FUNCTION_BLOCK FB_EstacionRestaurar_SFC
VAR_INPUT
    // SFC-Flags
    SFCPause: BOOL;
    SFCReset: BOOL;
    
    // Indicadores de sincronizacion
    Benido: BOOL := TRUE;
    Ejecuta: BOOL;
    
    // Entradas
    RechazadorDetras: BOOL; // Sobre el pale
    ManipuladorMedio: BOOL := TRUE; // En la vertical
    PrensadorArriba: BOOL := TRUE;
END_VAR
VAR_OUTPUT
    // Indicadores de sincronizacion
    Acabhe: BOOL;
    ListoKalisto: BOOL;
    
    // Salidas
    RechazadorRetrocede: BOOL; // Hacia el punto de trasvase de la prensa
END_VAR
VAR
END_VAR

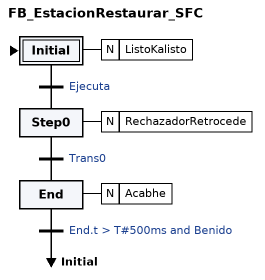
INITIAL_STEP Initial:
    ListoKalisto(N);
END_STEP
TRANSITION FROM Initial TO Step0
    := Ejecuta;
END_TRANSITION
STEP Step0:
    RechazadorRetrocede(N);
END_STEP
TRANSITION FROM Step0 TO End
    := Trans0;
END_TRANSITION
STEP End:
    Acabhe(N);
END_STEP
TRANSITION FROM End TO Initial
    := End.t > T#500ms and Benido;
END_TRANSITION

END_FUNCTION_BLOCK

(* stored: Version 1.1.0.1, ProductVersion 3.1.4024.12
   POU FB_EstacionRestaurar_SFC: Id {ce8cda89-3b60-43c8-b294-2c571b556ab8}, SpecialFunc None *)
